// TwinCAT 3 PLC project FMS_201_Manual
// ProgramVersion: 3.1.4023.0
// libraries:
//   CmpBitmapPool, * (System)
//   Tc2_Standard, * (Beckhoff Automation GmbH)
//   Tc2_System, * (Beckhoff Automation GmbH)
//   Tc3_Module, * (Beckhoff Automation GmbH)
//   VisuSymbols,3.5.10.0,System
// project tree:
//   / GlobalTextList.TcGTLO, PlcTask.TcTTO (not stored), Visualization Manager.TcVMO (not stored)
//   POUs/ FB_Estacion.TcPOU, MAIN.TcPOU, Vacio.TcIPO (not stored)
//   VISUs/ HMI_Proceso.TcVIS, Visualization.TcVIS (not stored)
// real-time tasks:
//   TASK PlcTask: cycle T#10ms, priority 20, ADS port 350
//   TASK PlcTask1: cycle T#10ms, priority 21, ADS port 351
//   TASK PlcTask2: cycle T#10ms, priority 22, ADS port 352
//   TASK PlcTask3: cycle T#10ms, priority 23, ADS port 353
//   TASK PlcTask4: cycle T#10ms, priority 24, ADS port 354
//   TASK PlcTask5: cycle T#10ms, priority 25, ADS port 355
//   TASK PlcTask6: cycle T#10ms, priority 26, ADS port 356
// I/O:
//   DEVICE Device 1 (EtherCAT), AmsNetId 5.67.250.180.2.1
//     Term 1 (EK1200) [EK1200-5000 EtherCAT Power supply (2A E-Bus)]
//       Term 2 (EL1008) [EL1008 8Ch. Dig. Input 24V, 3ms]
//       Term 3 (EL1008) [EL1008 8Ch. Dig. Input 24V, 3ms]
//       Term 4 (EL2008) [EL2008 8Ch. Dig. Output 24V, 0.5A]
//       Term 5 (EL2008) [EL2008 8Ch. Dig. Output 24V, 0.5A]
//       Term 6 (EL1008) [EL1008 8Ch. Dig. Input 24V, 3ms]
//       Term 7 (EL1008) [EL1008 8Ch. Dig. Input 24V, 3ms]
//       Term 8 (EL2008) [EL2008 8Ch. Dig. Output 24V, 0.5A]
//       Term 9 (EL2008) [EL2008 8Ch. Dig. Output 24V, 0.5A]
//       Term 10 (EL9011) [EL9011 End Terminal]
//   DEVICE Device 3 (RT-Ethernet Protocol), AmsNetId 5.67.250.180.4.1
//   DEVICE Device 2 (NOV-DP-RAM)
// variable links:
//   FMS_201_GEMMA/FMS_201_GEMMA Instance <-> Device 1 (EtherCAT)/Term 1 (EK1200)/Term 2 (EL1008)
//     PlcTask Inputs/MAIN.Estacion.EstacionConectada <-> Channel 5/EstacionConectada
//     PlcTask Inputs/MAIN.Estacion.PaleCodigoBit0 <-> Channel 7/PaleCodigoBit0
//     PlcTask Inputs/MAIN.Estacion.PaleCodigoBit1 <-> Channel 8/PaleCodigoBit1
//     PlcTask Inputs/MAIN.Estacion.PalePresencia <-> Channel 6/PalePresencia
//     PlcTask Inputs/MAIN.Estacion.PulsadorEmergencia <-> Channel 1/PulsadorEmergencia
//     PlcTask Inputs/MAIN.Estacion.PulsadorMarcha <-> Channel 3/PulsadorMarcha
//     PlcTask Inputs/MAIN.Estacion.PulsadorParada <-> Channel 4/PulsadorParada
//     PlcTask Inputs/MAIN.Estacion.SelectorManual <-> Channel 2/SelectorManual
//   FMS_201_GEMMA/FMS_201_GEMMA Instance <-> Device 1 (EtherCAT)/Term 1 (EK1200)/Term 3 (EL1008)
//     PlcTask Inputs/MAIN.Estacion.DetectorPresion <-> Channel 2/DetectorPresion
//     PlcTask Inputs/MAIN.Estacion.PaleCodigoBit2 <-> Channel 1/PaleCodigoBit2
//   FMS_201_GEMMA/FMS_201_GEMMA Instance <-> Device 1 (EtherCAT)/Term 1 (EK1200)/Term 4 (EL2008)
//     PlcTask Outputs/MAIN.Estacion.CintaMotorActiva <-> Channel 5/CintaMotorActiva
//     PlcTask Outputs/MAIN.Estacion.CintaMotorInvierte <-> Channel 6/CintaMotorInvierte
//     PlcTask Outputs/MAIN.Estacion.CintaRetenedorBaja <-> Channel 7/CintaRetenedorBaja
//     PlcTask Outputs/MAIN.Estacion.CintaSeparadorSube <-> Channel 8/CintaSeparadorSube
//     PlcTask Outputs/MAIN.Estacion.DesconectaEstacion <-> Channel 1/DesconectaEstacion
//     PlcTask Outputs/MAIN.Estacion.LamparaAlarma <-> Channel 2/LamparaAlarma
//     PlcTask Outputs/MAIN.Estacion.LamparaFaltaMaterial <-> Channel 4/LamparaFaltaMaterial
//     PlcTask Outputs/MAIN.Estacion.LamparaMarcha <-> Channel 3/LamparaMarcha
//   FMS_201_GEMMA/FMS_201_GEMMA Instance <-> Device 1 (EtherCAT)/Term 1 (EK1200)/Term 5 (EL2008)
//     PlcTask Outputs/MAIN.Estacion.AvisadorSonoro <-> Channel 1/AvisadorSonoro
//   FMS_201_GEMMA/FMS_201_GEMMA Instance <-> Device 1 (EtherCAT)/Term 1 (EK1200)/Term 6 (EL1008)
//     PlcTask Inputs/MAIN.Estacion.AlimentadorDetras <-> Channel 8/AlimentadorDetras
//     PlcTask Inputs/MAIN.Estacion.DescargadorDelante <-> Channel 2/DescargadorDelante
//     PlcTask Inputs/MAIN.Estacion.DescargadorDetras <-> Channel 1/DescargadorDetras
//     PlcTask Inputs/MAIN.Estacion.DesplazadorDetras <-> Channel 7/DesplazadorDetras
//     PlcTask Inputs/MAIN.Estacion.VerificadorAbajo <-> Channel 6/VerificadorAbajo
//     PlcTask Inputs/MAIN.Estacion.VerificadorArriba <-> Channel 5/VerificadorArriba
//     PlcTask Inputs/MAIN.Estacion.VerticalAbajo <-> Channel 4/VerticalAbajo
//     PlcTask Inputs/MAIN.Estacion.VerticalArriba <-> Channel 3/VerticalArriba
//   FMS_201_GEMMA/FMS_201_GEMMA Instance <-> Device 1 (EtherCAT)/Term 1 (EK1200)/Term 7 (EL1008)
//     PlcTask Inputs/MAIN.Estacion.AlimentadorDelante <-> Channel 1/AlimentadorDelante
//     PlcTask Inputs/MAIN.Estacion.PresenciaBaseAlimentador <-> Channel 3/PresenciaBaseAlimentador
//     PlcTask Inputs/MAIN.Estacion.VacioDescargador <-> Channel 2/VacioDescargador
//   FMS_201_GEMMA/FMS_201_GEMMA Instance <-> Device 1 (EtherCAT)/Term 1 (EK1200)/Term 8 (EL2008)
//     PlcTask Outputs/MAIN.Estacion.AlimentadorAdelante <-> Channel 7/AlimentadorAdelante
//     PlcTask Outputs/MAIN.Estacion.DescargadorAdelante <-> Channel 1/DescargadorAdelante
//     PlcTask Outputs/MAIN.Estacion.DescargadorAtras <-> Channel 2/DescargadorAtras
//     PlcTask Outputs/MAIN.Estacion.DescargadorBaja <-> Channel 3/DescargadorBaja
//     PlcTask Outputs/MAIN.Estacion.DesplazadorAdelante <-> Channel 6/DesplazadorAdelante
//     PlcTask Outputs/MAIN.Estacion.EyectorSucciona <-> Channel 8/EyectorSucciona
//     PlcTask Outputs/MAIN.Estacion.RechazadorAdelante <-> Channel 4/RechazadorAdelante
//     PlcTask Outputs/MAIN.Estacion.VerificadorBaja <-> Channel 5/VerificadaorBaja

// ---- POUs/FB_Estacion.TcPOU
FUNCTION_BLOCK FB_Estacion
VAR_INPUT
END_VAR
VAR_OUTPUT
	//Parametros de salida
	PaleCodigo: BYTE;
END_VAR
VAR
	//Entradas comunes
	PulsadorEmergencia AT %I*: BOOL;
    SelectorManual AT %I*: BOOL;
    PulsadorMarcha AT %I*: BOOL;
    PulsadorParada AT %I*: BOOL := TRUE; // Contacto normalmente cerrado
    EstacionConectada AT %I*: BOOL := TRUE;
    DetectorPresion AT %I*: BOOL := TRUE;
	
	PalePresencia AT %I*: BOOL;
    PaleCodigoBit0 AT %I*: BOOL;
    PaleCodigoBit1 AT %I*: BOOL;
    PaleCodigoBit2 AT %I*: BOOL;
	
	//Entradas específicas
	DescargadorDetras AT %I*: BOOL;
	DescargadorDelante AT %I*: BOOL;
	VerticalArriba AT %I*: BOOL;
	VerticalAbajo AT %I*: BOOL;
	VerificadorArriba AT %I*: BOOL;
	VerificadorAbajo AT %I*: BOOL;
	DesplazadorDetras AT %I*: BOOL;
	AlimentadorDetras AT %I*: BOOL;
	AlimentadorDelante AT %I*: BOOL;
	VacioDescargador AT %I*: BOOL;
	PresenciaBaseAlimentador AT %I*:BOOL;
	
	//Salidas comunes
	DesconectaEstacion AT %Q*: BOOL;
    LamparaAlarma AT %Q*: BOOL;
    LamparaMarcha AT %Q*: BOOL;
	LamparaFaltaMaterial AT %Q*: BOOL;
    AvisadorSonoro AT %Q*: BOOL;

    CintaMotorActiva AT %Q*: BOOL;
    CintaMotorInvierte AT %Q*: BOOL;
    CintaRetenedorBaja AT %Q*: BOOL;
    CintaSeparadorSube AT %Q*: BOOL;
	
	//Salidas específicas
	DescargadorAtras AT %Q*: BOOL;
	DescargadorAdelante AT %Q*: BOOL;
	DescargadorBaja AT %Q*: BOOL;
	RechazadorAdelante AT %Q*: BOOL;
	VerificadorBaja AT %Q*: BOOL;
	DesplazadorAdelante AT %Q*: BOOL;
	AlimentadorAdelante AT %Q*: BOOL;
	EyectorSucciona AT %Q*: BOOL;
END_VAR

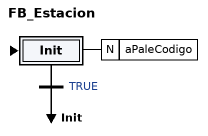
INITIAL_STEP Init:
    aPaleCodigo(N);
END_STEP
TRANSITION FROM Init TO Init
    := TRUE;
END_TRANSITION

ACTION aPaleCodigo:
PaleCodigo.0 := PaleCodigoBit0;
PaleCodigo.1 := PaleCodigoBit1;
PaleCodigo.2 := PaleCodigoBit2;
END_ACTION

END_FUNCTION_BLOCK

// ---- POUs/MAIN.TcPOU
PROGRAM MAIN
VAR
	ESTACION: FB_Estacion;
END_VAR

ESTACION();

END_PROGRAM

// ---- GlobalTextList.TcGTLO
TEXTLIST GlobalTextList
  699 = '%d'
  788 = 'A+'
  680 = 'A-'
  976 = 'ALARMA'
  736 = 'ALIMENTACIÓN DE LA BASE'
  789 = 'Alimentador '
  282 = 'Alimentador adelante'
  826 = 'ALIMENTADOR DE TAPAS'
  339 = 'ALIMENTADORA DE BASES'
  91 = 'ALIMENTAR'
  778 = 'B+'
  544 = 'B-'
  615 = 'Chupar'
  903 = 'Descargador\n Adelante'
  271 = 'Descargador\n Atras'
  14 = 'Descargador\n Atrás'
  363 = 'Descargador\n Descargador\nVertical'
  695 = 'Descargador\nVertical'
  296 = 'Descargador /n Adelante'
  174 = 'Descargador Adelante'
  200 = 'Descargador \\n Adelante'
  816 = 'DescargadorAdelante'
  467 = 'DescargadorAdelante\nHola'
  386 = 'Descargador\\n Adelante'
  53 = 'Desplazador\nadelante'
  32 = 'DESPLAZAR'
  872 = 'Detector\nPresion'
  471 = 'E+'
  179 = 'E-'
  895 = 'F+'
  802 = 'F-'
  399 = 'FMS 201'
  707 = 'FMS-201'
  652 = 'FMS-201\t\tALIMENTACIÓN DE LA BASE'
  847 = 'Manual'
  727 = 'MARCHA'
  958 = 'MATERIAL'
  646 = 'Nº PALE'
  999 = 'OFF'
  328 = 'OK'
  374 = 'ON'
  582 = 'Pale\nPresencia'
  284 = 'Pulsador\nEmergencia'
  820 = 'Pulsador\nMarcha'
  285 = 'Pulsador\nParada'
  165 = 'Pulsador Emergencia'
  392 = 'RETENEDOR'
  252 = 'Selector\nManual'
  585 = 'SEPARADOR'
  442 = 'SUCCIONAR'
  391 = 'V+'
  726 = 'VERIFICAR'
  661 = 'x'
END_TEXTLIST

// ---- VISUs/HMI_Proceso.TcVIS
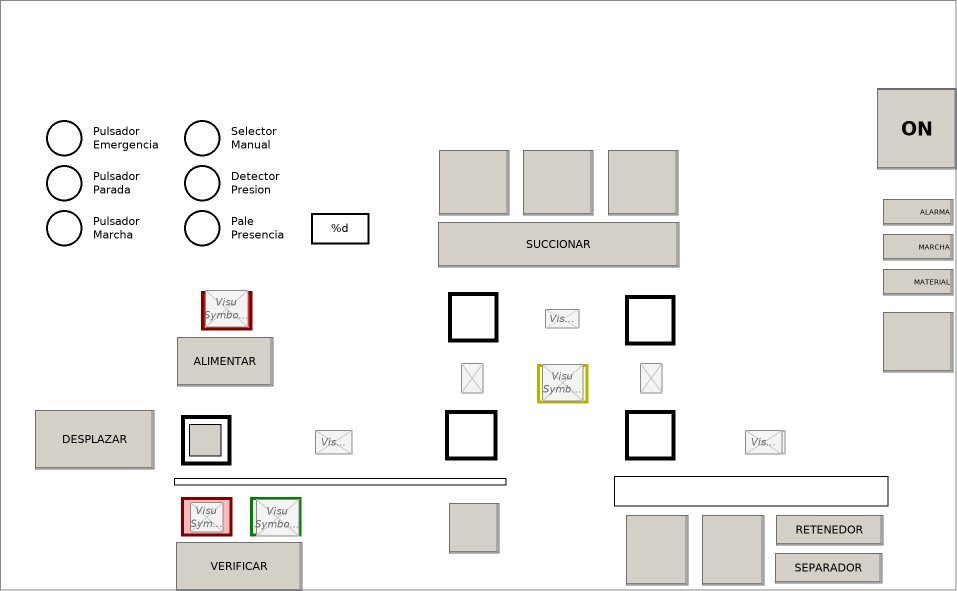
VISUALIZATION HMI_Proceso  // 957x591
    Rectangle (174,478 332x7)
    Rectangle (614,476 274x30)
    Button (176,542 126x49), "VERIFICAR"
        toggle MAIN.ESTACION.VerificadorBaja
    RoundedRectangle (250,497 51x39), colour toggle: MAIN.ESTACION.VerificadorAbajo
    RoundedRectangle (181,497 51x39), colour toggle: MAIN.ESTACION.VerificadorArriba
    Button (449,503 50x50), image: VisuSymbols.Symbols.Delete
        tap MAIN.ESTACION.RechazadorAdelante
    Image (256,499 43x37), image: VisuSymbols.Symbols.OK
    Image (190,502 33x30), image: VisuSymbols.Symbols.Wrong
    Button (35,410 119x59), "DESPLAZAR"
        toggle MAIN.ESTACION.DesplazadorAdelante
    Rectangle (445,410 52x50)
        p4110469609: SEL(MAIN.ESTACION.DescargadorDetras AND MAIN.ESTACION.VerticalAbajo, 2, 0)
    Rectangle (181,415 50x50)
        p4110469609: SEL(MAIN.ESTACION.DesplazadorDetras, 2, 0)
    Rectangle (448,292 50x50)
        p4110469609: SEL((MAIN.ESTACION.DescargadorDetras AND MAIN.ESTACION.VerticalArriba), 2, 0)
    Rectangle (625,295 50x50)
        p4110469609: SEL(MAIN.ESTACION.DescargadorDelante AND MAIN.ESTACION.VerticalArriba, 2, 0)
    Rectangle (625,410 50x50)
        p4110469609: SEL(MAIN.ESTACION.DescargadorDelante AND MAIN.ESTACION.VerticalAbajo, 2, 0)
    Button (438,222 241x45), "SUCCIONAR"
        toggle MAIN.ESTACION.EyectorSucciona
    Button (439,150 70x65), image: VisuSymbols.Symbols.TriangleLeft
        tap MAIN.ESTACION.DescargadorAtras
    Button (523,150 70x65), image: VisuSymbols.Symbols.TriangleDown
        toggle MAIN.ESTACION.DescargadorBaja
    Button (608,150 70x65), image: VisuSymbols.Symbols.TriangleRight
        tap MAIN.ESTACION.DescargadorAdelante
    Image (545,309 34x19), image: VisuSymbols.Symbols.DoubleArrow3
    Image (640,363 22x30), image: VisuSymbols.Symbols.DoubleArrow4
    Image (461,363 22x30), image: VisuSymbols.Symbols.DoubleArrow4
    Image (315,430 37x24), image: VisuSymbols.Symbols.ArrowBoldRight
    Image (748,430 37x24), invisible if: MAIN.ESTACION.CintaMotorInvierte, image: VisuSymbols.Symbols.ArrowBoldRight
    RoundedRectangle (201,291 51x39), colour toggle: MAIN.ESTACION.PresenciaBaseAlimentador
    RoundedRectangle (537,364 51x39), colour toggle: MAIN.ESTACION.VacioDescargador
    Image (542,364 41x37), image: VisuSymbols.Symbols.Caution
    Rectangle (190,425 30x30), invisible if: not(main.ESTACION.AlimentadorDelante)
    Image (216,296 24x30), invisible if: MAIN.ESTACION.PresenciaBaseAlimentador, image: Vacio.vacio
    Button (626,515 62x70), image: Vacio.onoff
        toggle MAIN.ESTACION.CintaMotorActiva
    Button (702,515 62x70), image: VisuSymbols.Symbols.ArrowCircle2RightUpDown
        toggle MAIN.ESTACION.CintaMotorInvierte
    Button (776,515 107x30), "RETENEDOR"
        toggle MAIN.ESTACION.CintaRetenedorBaja
    Button (775,553 107x30), "SEPARADOR"
        toggle MAIN.ESTACION.CintaSeparadorSube
    Image (205,290 43x37), invisible if: not(main.ESTACION.PresenciaBaseAlimentador), image: VisuSymbols.Symbols.OK
    Button (877,88 80x80), "OFF", invisible if: MAIN.ESTACION.EstacionConectada
    Button (883,199 70x26), "ALARMA", image: VisuSymbols.Symbols.light
        toggle MAIN.ESTACION.LamparaAlarma
    Button (883,234 70x26), "MARCHA", image: VisuSymbols.Symbols.light
        toggle MAIN.ESTACION.LamparaMarcha
    Button (883,269 70x26), "MATERIAL", image: VisuSymbols.Symbols.light
        toggle MAIN.ESTACION.LamparaFaltaMaterial
    Button (883,312 70x60), image: VisuSymbols.Symbols.loudspeakerMedium
        toggle MAIN.ESTACION.AvisadorSonoro
    Rectangle (189,424 32x32), invisible if: (not(MAIN.ESTACION.AlimentadorDetras) OR not(main.ESTACION.PresenciaBaseAlimentador))
    Button (177,337 96x49), "ALIMENTAR"
        toggle MAIN.ESTACION.AlimentadorAdelante
    Button (877,89 80x80), "ON", invisible if: NOT MAIN.ESTACION.EstacionConectada
        tap MAIN.ESTACION.DesconectaEstacion
    Ellipse (46,120 36x36), colour toggle: MAIN.ESTACION.PulsadorEmergencia
    Ellipse (46,165 36x36), colour toggle: not(MAIN.ESTACION.PulsadorParada)
    Ellipse (46,210 36x36), colour toggle: MAIN.ESTACION.PulsadorMarcha
    Ellipse (184,120 36x36), colour toggle: MAIN.ESTACION.SelectorManual
    Ellipse (184,165 36x36), colour toggle: MAIN.ESTACION.DetectorPresion
    Label (90,123 83x30), "Pulsador Emergencia"
    Label (90,168 83x30), "Pulsador Parada"
    Label (90,213 83x30), "Pulsador Marcha"
    Label (228,123 83x30), "Selector Manual"
    Label (228,168 83x30), "Detector Presion"
    Ellipse (184,210 36x36), colour toggle: MAIN.ESTACION.PalePresencia
    Label (228,213 83x30), "Pale Presencia"
    Rectangle (311,213 58x31), "%d", text variable: MAIN.ESTACION.PaleCodigo, invisible if: not(MAIN.ESTACION.PalePresencia)
    Image (745,430 37x24), invisible if: not(MAIN.ESTACION.CintaMotorInvierte), image: VisuSymbols.Symbols.ArrowBoldLeft
END_VISUALIZATION
